// TIA Portal V18 export
DATA_BLOCK "MES_CheckControl"   // DB2361
{ S7_Optimized_Access := 'FALSE' }
VERSION : 0.1
// stored: AutoNumber false, DBAccessibleFromOPCUA true, DBAccessibleFromWebserver true, IsOnlyStoredInLoadMemory false, IsWriteProtectedInAS false
   VAR
      ST1MesCheckIn : Bool;
      ST1MesCheckOut : Bool;
      ST2MesCheckIn : Bool;
      ST2MesCheckOut : Bool;
      ST3MesCheckIn : Bool;
      ST3MesCheckOut : Bool;
      ST4MesCheckIn : Bool;
      ST4MesCheckOut : Bool;
      Station1 : Struct
         CheckInRequest : Bool;
         CheckResultRequest : Bool;
      END_STRUCT;
      Station2 : Struct
         CheckInRequest : Bool;
         CheckResultRequest : Bool;
      END_STRUCT;
      Station3 : Struct
         CheckInRequest : Bool;
         CheckResultRequest : Bool;
      END_STRUCT;
      Station4 : Struct
         CheckInRequest : Bool;
         CheckResultRequest : Bool;
      END_STRUCT;
      Station5 : Struct
         CheckInRequest : Bool;
         CheckResultRequest : Bool;
      END_STRUCT;
      Station6 : Struct
         CheckInRequest : Bool;
         CheckResultRequest : Bool;
      END_STRUCT;
      Station7 : Struct
         CheckInRequest : Bool;
         CheckResultRequest : Bool;
      END_STRUCT;
   END_VAR
BEGIN
END_DATA_BLOCK
